TYPE ELL6AttenuationFilterConfig EXTENDS DeviceConfiguration :
STRUCT
	SerialCommunication : SerialCommunication;
END_STRUCT
END_TYPE

(* stored: Version 1.1.0.1, ProductVersion 3.1.4024.10
   DUT ELL6AttenuationFilterConfig: Id {33d3baa2-bb2e-4cf6-a935-346765a625a5} *)
